// Mitsubishi GX Works2 project: NOT   PLC: Q03UDV

PROGRAM MAIN
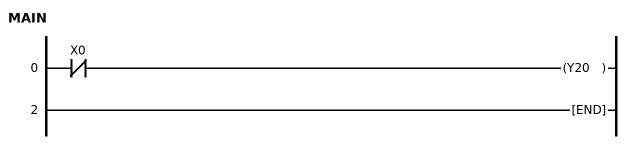
0     LDI     X0
      OUT     Y20
2     END
END_PROGRAM
